ABB RobotStudio station: Lab1_4_20210903-134352.rsstn

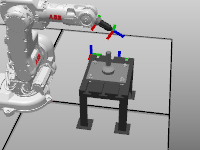
Station Lab1_4 (saved by RobotStudio 21.2.9526.0)
Layout (positions relative to the parent item):
  - IRB140_6_81_C_03 [mechanism, from Robots\IRB140_6_81_C_G_03.rslib] at (0, 0, 0) mm; joint values [0, 0, 0, 0, 0.5236, 0] (rad or m)
  - UISpenholder [mechanism, from RS1\UISpenholder.rslib] at (506.29, 0, 679.5) mm, rotated rx 180 ry 60 rz 180 deg
  - table_and_fixture_140 [part, from Training Objects\propeller_table.rslib] at (400, 220, 0) mm, rotated rx 0 ry 0 rz -90 deg
Attachment: UISpenholder is attached to IRB140_6_81_C_03 / Link6
Attachment: WobjTable is attached to table_and_fixture_140
Targets, tools, work objects and paths stored in the station, written as RAPID:
! task (no controller)
MODULE CalibData
  TASK PERS wobjdata WobjTable:=[FALSE,TRUE,"",[[575,620,0],[0.707106781,0,0,-0.707106781]],[[425,-150,308],[1,0,0,0]]];
ENDMODULE

! task (no controller)
MODULE CalibData
  PERS tooldata UISpenholder:=[TRUE,[[0,0,110],[1,0,0,0]],[1,[0,0,1],[1,0,0,0],0,0,0]];
ENDMODULE

